PROGRAM MAIN

VAR
	{attribute 'OPC.UA.DA' := '1'}
	FB_DMXDiscovery512_01: FB_DMXDiscovery512;
	{attribute 'OPC.UA.DA' := '1'}
	DMX_CommandBuffer:ST_DMXCommandBuffer;
	FB_EL6851CommunicationEx_01: FB_EL6851CommunicationEx;
	ST_EL6851InData_01 AT %I* : ST_EL6851InDataEx;
	ST_EL6851OutData_01 AT %Q*: ST_EL6851OutData;
	ProcessData : ARRAY [1..512] OF BYTE; 
	{attribute 'OPC.UA.DA' := '1'}
	Mover1 AT %Q* : Mover_13Ch;
	
	{attribute 'OPC.UA.DA' := '1'}
	FixtureChLength : UINT := 13;
	
	{attribute 'OPC.UA.DA' := '1'}
	TestBool : BOOL;
	
END_VAR



(*FB_EL6851CommunicationEx_01(
	wSourceManufacturerId:= , 
	dwSourceDeviceId:= , 
	bEnableSendingData:= , 
	bSetCycleMode:= , 
	bSendDefaultData:= , 
	uiDataLength:= , 
	dwOptions:= , 
	bError=> , 
	udiErrorId=> , 
	bCycleMode=> , 
	byBufferDemandMeter=> , 
	byBufferMaximumDemandMeter=> , 
	uiBufferOverflowCounter=> , 
	bLineIsBusy=> , 
	stEL6851InData:= ST_EL6851InData_01, 
	stEL6851OutData:= ST_EL6851OutData_01, 
	stCommandBuffer:= DMX_CommandBuffer, 
	arrProcessData:= ProcessData);


FB_DMXDiscovery512_01(
	bStart:= , 
	dwOptions:= DMX_OPTION_COMPLETE_NEW_DISCOVERY, 
	bBusy=> , 
	bError=> , 
	udiErrorId=> , 
	uliLowerBoundSearchUID=> , 
	uliUpperBoundSearchUID=> , 
	arrDMXDeviceInfoList=> , 
	uiNextDMX512StartAddress=> , 
	iFoundDevices=> , 
	stCommandBuffer:= DMX_CommandBuffer);
*)

END_PROGRAM

(* stored: Version 1.1.0.1
   POU MAIN: Id {5b7ed463-4ea7-4cdb-807c-6eeb36d90ee8}, SpecialFunc None *)
